// TIA Portal V17 export
// export: Created 2024-08-29T18:23:49.4121976Z, ExportSetting WithDefaults, DisplayName Totally Integrated Automation Portal, DisplayVersion V17 Update 7, DisplayName TIA Portal Openness, DisplayVersion V17 Update 7, DisplayName TIA Portal Version Control Interface, DisplayVersion V17, DisplayName SINAMICS Startdrive Advanced, DisplayVersion V17 SP2, DisplayName SINAMICS Startdrive G110M, G120, G120C, G120D, G120P, G115D, DisplayVersion V17 SP2, DisplayName SINAMICS Startdrive G130, G150, S120, S150, SINAMICS MV, S210, DisplayVersion V17 SP2, DisplayName STEP 7 Professional, DisplayVersion V17 Update 7, DisplayName STEP 7 Safety, DisplayVersion V17 Update 6, DisplayName WinCC Advanced / Unified PC, DisplayVersion V17 Update 7
DATA_BLOCK "Port_Config_DB2"   // DB38
// stored: AutoNumber true, DBAccessibleFromOPCUA true, DBAccessibleFromWebserver true, InstanceOfName Port_Config, OfSystemLibElement Port_Config, OfSystemLibVersion 1.2
"Port_Config"
   // VAR_INPUT
   //    REQ : Bool := TRUE;
   //    PORT : PORT := 284;
   //    PROTOCOL : UInt := 0;
   //    BAUD : UInt := 6;
   //    PARITY : UInt := 1;
   //    DATABITS : UInt := 1;
   //    STOPBITS : UInt := 1;
   //    FLOWCTRL : UInt := 2;
   //    XONCHAR : Char := '$0B';
   //    XOFFCHAR : Char := '$R';
   //    WAITTIME : UInt := 2000;
   //    MODE : USInt := 0;
   //    LINE_PRE : USInt := 0;
   //    BRK_DET : USInt := 0;
   // END_VAR
   // VAR_OUTPUT
   //    DONE : Bool := FALSE;
   //    ERROR : Bool := FALSE;
   //    STATUS : Word := 16#7000;
   // END_VAR
   // VAR
   //    b_e_REQ : Bool := TRUE;
   //    y_state : SInt := 0;
   //    WRREC { S7_SetPoint := 'True'} : WRREC;
   //    RDREC { S7_SetPoint := 'True'} : RDREC;
   //    w_record { S7_SetPoint := 'True'} : P2P_PortData;
   //    r_record { S7_SetPoint := 'True'} : P2P_RdEstat;
   // END_VAR
BEGIN
   WRREC.REQ := FALSE;
   WRREC.ID := 284;
   WRREC.INDEX := 57;
   WRREC.LEN := 28;
   WRREC.DONE := TRUE;
   WRREC.BUSY := FALSE;
   WRREC.ERROR := FALSE;
   WRREC.STATUS := 16#0000_0000;
   RDREC.REQ := FALSE;
   RDREC.ID := 0;
   RDREC.INDEX := 0;
   RDREC.MLEN := 0;
   RDREC.VALID := FALSE;
   RDREC.BUSY := FALSE;
   RDREC.ERROR := FALSE;
   RDREC.STATUS := 16#0000_0000;
   RDREC.LEN := 0;
   w_record.header.block_type := 16#0039;
   w_record.header.block_len := 16#0018;
   w_record.header.block_ver := 16#0100;
   w_record.header.res := 16#0000;
   w_record.PROTOCOL := 0;
   w_record.BAUD := 6;
   w_record.PARITY := 1;
   w_record.DATABITS := 1;
   w_record.STOPBITS := 1;
   w_record.FLOWCTRL := 2;
   w_record.XONCHAR := '$0B';
   w_record.XOFFCHAR := '$R';
   w_record.WAITTIME := 2000;
   w_record.MODE := 0;
   w_record.LINE_PRE := 0;
   w_record.BRK_DET := 0;
   w_record.LibSupport := 16#00;
   w_record.res := 16#00;
   r_record.header.block_type := 16#0000;
   r_record.header.block_len := 16#0000;
   r_record.header.block_ver := 16#0000;
   r_record.header.res := 16#0000;
   r_record.SetFtrs := 16#0000;
   r_record.PortCfg := 16#0000;
   r_record.SendCfg := 16#0000;
   r_record.RcvCfg := 16#0000;
   r_record.SgnSet := 16#0000;
   r_record.R3964Err := 16#0000;
END_DATA_BLOCK
